FUNCTION_BLOCK AR_CALIBRATE_2P_REF (* Adapter-based 2-point calibration (Low/High, independently stored - no CO-before-CS style ordering dependency) - reference targets (Y_LOW/Y_HIGH) are live AR sockets, persisted via 2 additional AR2 plugs (LOW_REF/HIGH_REF), same live-echo pattern as AR_CALIBRATE_SQ_REF *)
  (* Standard: 61499-1 *)
  (* Version 1.3, 2026-09-21, Franz Höpfinger, Code-Review-Fund (PR #260): xClipping clippte bisher unconditional auf [LOW_REF,HIGH_REF], auch wenn nur EIN Punkt kalibriert war - der jeweils andere, noch unkalibrierte Referenzwert stand dann noch auf seinem INI_AR2-Default 0.0, wodurch der frisch eingefuehrte Partial-Kalibrierung-Fallback (Y.D1 := LOW_REF.DI1 bzw. HIGH_REF.DI1) sofort wieder auf 0.0 zurueckgeklemmt wurde - der Wert griff also weiterhin nicht sofort. Clipping jetzt zusaetzlich an xLowCal AND xHighCal gegated. *)
  (* Version 1.2, 2026-09-21, Franz Höpfinger, Genauso geaendert wie AR_CALIBRATE_3P_REF: INIT/QI/QO/INITO-Pattern (Enable/Disable) ergaenzt. Neuer Input xClipping (Default TRUE) - bisher clippte dieser Typ ueberhaupt nicht, jetzt optional auf LOW_REF..HIGH_REF klemmbar (FALSE = altes Verhalten, keine Klemmung). Neue interne Kalibriert-Flags xLowCal/xHighCal (latchen TRUE, sobald der jeweilige Rohwert vom INI_AR2-Default 0.0 abweicht): solange nur EIN Punkt kalibriert ist, wurde bisher trotzdem interpoliert - gegen einen Rohwert-Default von 0.0 fuer den jeweils anderen, noch unkalibrierten Punkt, was ein Garbage-Ergebnis lieferte. Jetzt liefert REQ in diesem Fall stattdessen direkt den REF-Wert des einen kalibrierten Punkts. *)
  (* Version 1.1, 2026-09-17, Franz Höpfinger, C_LOW/C_HIGH von AX-Sockets (mit [C_LOW.D1]/[C_HIGH.D1]-Flankenwaechter) auf reine EventInputs umgestellt - Franz: jeder echte Aufrufer (VT-Taste, OPC-UA-Methode, Remote-Toggle-Trigger nach Merge) liefert ohnehin ein atomares, einmaliges Event, der D1-Wert war bei jedem tatsaechlichen Caller immer hartcodiert TRUE (via AX_BOOL_TO_X) und der Guard filterte nie etwas - reine akademische Rechtfertigung ohne echten Nutzen. Aufrufer muessen jetzt direkt ein Event statt eines AX-Adapters anschliessen (AX_BOOL_TO_X-Umweg entfaellt). *)
  (* Version 1.0, 2026-09-11, Meisterschulen am Ostbahnhof, Ersatz fuer AR_CALIBRATE_SQ_REF: dieselbe Formel/dasselbe Ergebnis, aber ohne die CO-vor-CS-Abhaengigkeit - jeder Punkt speichert unabhaengig seinen Rohwert (wie AR_CALIBRATE_3P), die Interpolation passiert erst live bei X.E1, nicht mehr inkrementell beim Kalibrieren selbst. *)
  PACKAGE adapter::Engineering::measurements;
  (* Documentation:
  Formula
   Y = LOW_REF + (X - X_LOW) * (HIGH_REF - LOW_REF) / (X_HIGH - X_LOW), clipped to LOW_REF..HIGH_REF unless xClipping = FALSE Partial Calibration (before both points are set)
   Each point is tracked internally (xLowCal/xHighCal, latched TRUE once its raw value differs from the INI_AR2 default 0.0). Until both are calibrated, REQ falls back to the one already-known REF value instead of interpolating against the other point's still-0.0 default (which previously produced a garbage result as soon as only one side had been calibrated).
   Why this replaces AR_CALIBRATE_SQ_REF
   AR_CALIBRATE_SQ_REF computes OFFSET/SCALE incrementally (CO sets OFFSET from a live SCALE, CS then recomputes both from an internal X_LOW_INT/Y_LOW_INT captured by CO) - CS is only mathematically valid after CO has run at least once, which needed an ECC-enforced order to avoid a silent garbage-OFFSET calibration.
   This type stores X_LOW/X_HIGH completely independently (exactly like AR_CALIBRATE_3P/AR_CALIBRATE_3P_REF store X_MIN/X_MID/X_MAX) and only combines them into a line at read-time (REQ), which runs on every X.E1 regardless of calibration state. There is no data dependency between C_LOW and C_HIGH, so there is nothing an enforced order could protect against - both points can be (re-)calibrated in any order, independently, at any time.
   Calibration (Two-Point, Free Order)
    - Low (C_LOW): Apply low reference, set Y_LOW to desired output, trigger C_LOW → X_LOW := X
   - High (C_HIGH): Apply high reference, set Y_HIGH to desired output, trigger C_HIGH → X_HIGH := X
    Either point can be recalibrated on its own at any later time (e.g. re-trimming a drifted zero point) without repeating the other.
   Reference Targets (Y_LOW / Y_HIGH) are live AR Sockets
   Same live-echo mechanism as AR_CALIBRATE_SQ_REF: Y_LOW/Y_HIGH are bidirectional AR2 Sockets fed from an external VT/web reader, mirrored out through the AR2 Plugs LOW_REF/HIGH_REF for persistence (INI_AR2/NVS_AR2), and echoed back via LOW_REF.EI1/HIGH_REF.EI1 so a boot-restored value shows up on screen without the operator re-entering it.
  *)
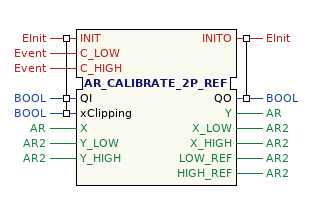
  EVENT_INPUT
    INIT : EInit WITH QI, xClipping; (* Initialization Request *)
    C_LOW; (* Calibrate Low Point - atomarer Trigger (VT-Taste/OPC-UA-Methode/Remote-Toggle nach Merge) *)
    C_HIGH; (* Calibrate High Point - atomarer Trigger (VT-Taste/OPC-UA-Methode/Remote-Toggle nach Merge) *)
  END_EVENT
  EVENT_OUTPUT
    INITO : EInit WITH QO; (* Initialization Confirm *)
  END_EVENT
  VAR_INPUT
    QI : BOOL; (* Input event qualifier *)
    xClipping : BOOL := TRUE; (* TRUE (Default) = Ausgang wird auf LOW_REF..HIGH_REF geklemmt; FALSE = kein Clipping, Extrapolation ueber die Kalibrierpunkte hinaus erlaubt (bisheriges Verhalten) *)
  END_VAR
  VAR_OUTPUT
    QO : BOOL; (* Output event qualifier *)
  END_VAR
  SOCKETS
    X : adapter::types::unidirectional::AR; (* Raw Input *)
    Y_LOW : adapter::types::bidirectional::AR2; (* Target output Y at the low calibration point - live edit in via EO1/DO1 (Socket-side swap), persisted/restored value echoed back out via EI1/DI1 for VT/web display *)
    Y_HIGH : adapter::types::bidirectional::AR2; (* Target output Y at the high calibration point - live edit in via EO1/DO1 (Socket-side swap), persisted/restored value echoed back out via EI1/DI1 for VT/web display *)
  END_SOCKETS
  PLUGS
    Y : adapter::types::unidirectional::AR; (* Calibrated Output *)
    X_LOW : adapter::types::bidirectional::AR2; (* Persisted raw input value at the low calibration point *)
    X_HIGH : adapter::types::bidirectional::AR2; (* Persisted raw input value at the high calibration point *)
    LOW_REF : adapter::types::bidirectional::AR2; (* Persisted low-point target reference (Y_LOW) *)
    HIGH_REF : adapter::types::bidirectional::AR2; (* Persisted high-point target reference (Y_HIGH) *)
  END_PLUGS
  VAR
    xLowCal : BOOL := FALSE; (* Latched TRUE sobald X_LOW.DI1 vom INI-Default 0.0 abweicht - LOW wurde mindestens einmal kalibriert (diese Session oder ueber Boot-Restore) *)
    xHighCal : BOOL := FALSE; (* Latched TRUE sobald X_HIGH.DI1 vom INI-Default 0.0 abweicht - HIGH wurde mindestens einmal kalibriert (diese Session oder ueber Boot-Restore) *)
  END_VAR
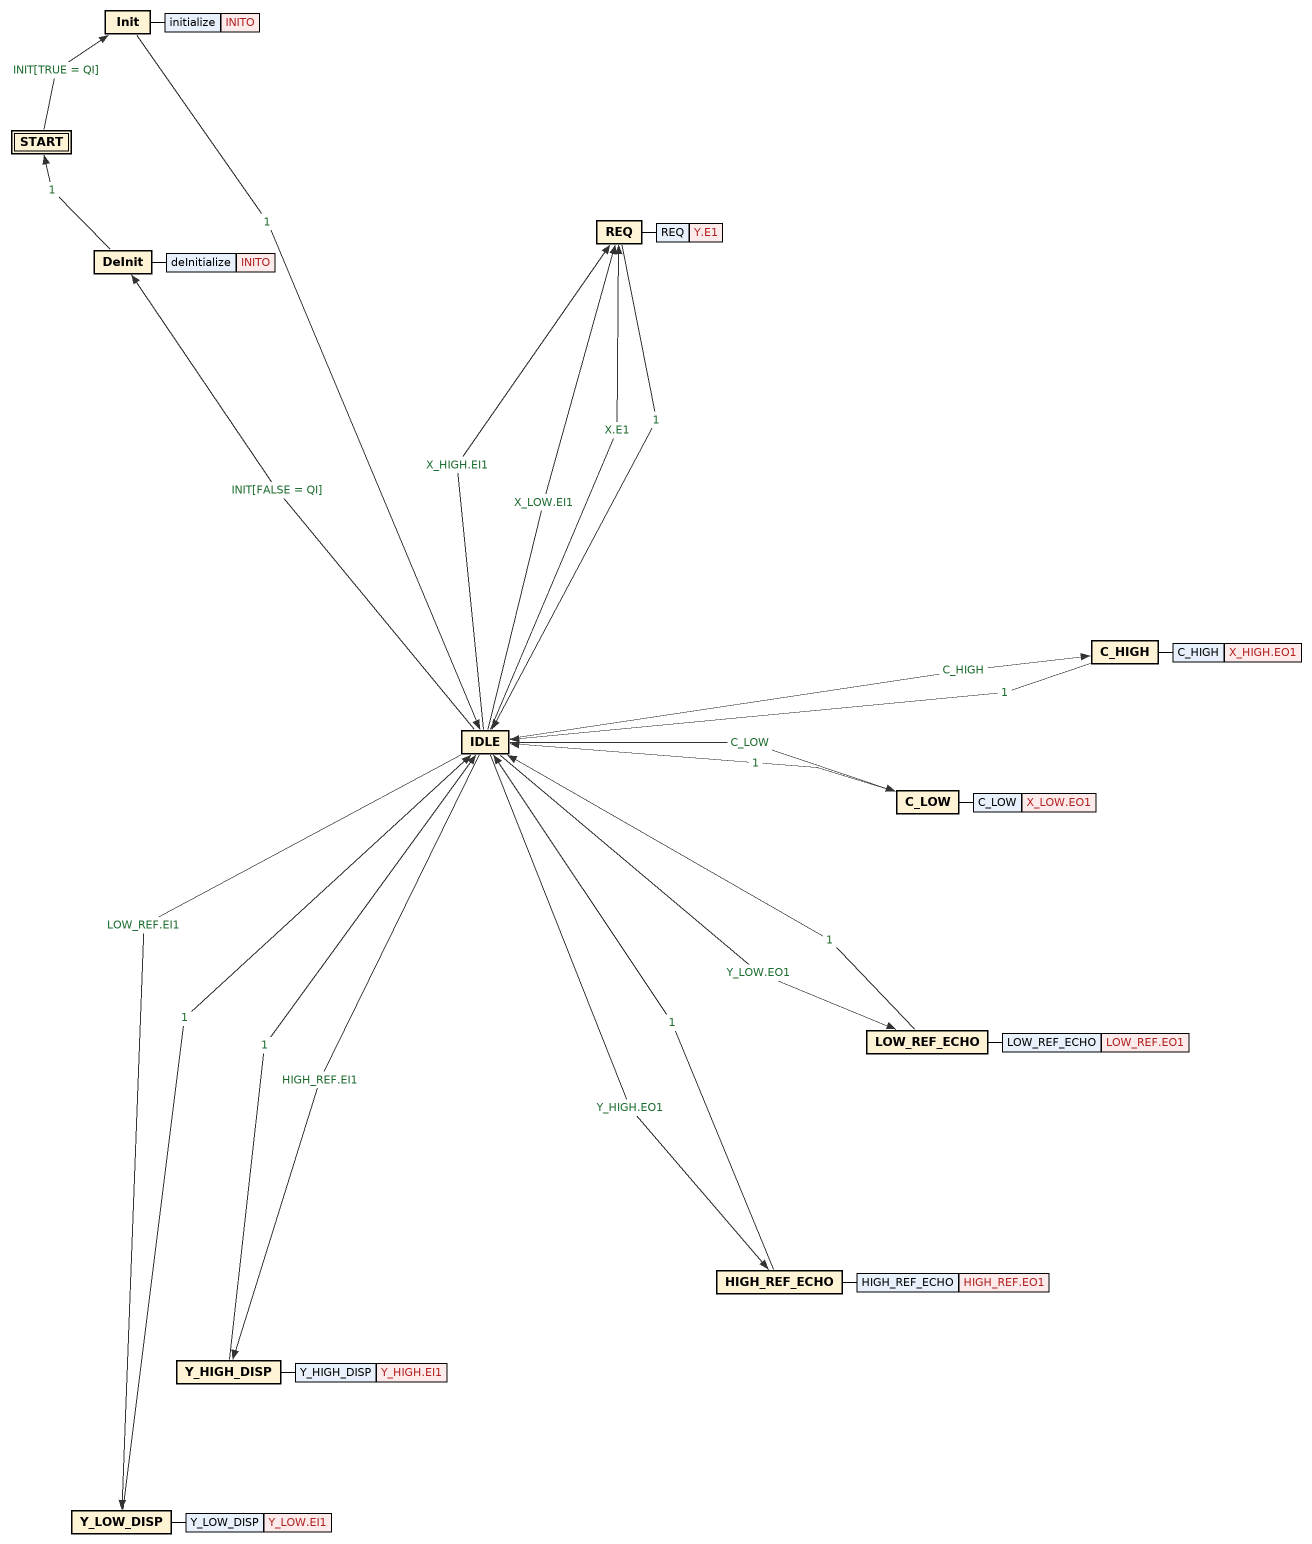
  EC_STATES
    START; (* Initial State *)
    Init : initialize -> INITO; (* Initialization *)
    DeInit : deInitialize -> INITO;
    IDLE;
    REQ : REQ -> Y.E1;
    C_LOW : C_LOW -> X_LOW.EO1;
    C_HIGH : C_HIGH -> X_HIGH.EO1;
    LOW_REF_ECHO : LOW_REF_ECHO -> LOW_REF.EO1;
    HIGH_REF_ECHO : HIGH_REF_ECHO -> HIGH_REF.EO1;
    Y_LOW_DISP : Y_LOW_DISP -> Y_LOW.EI1;
    Y_HIGH_DISP : Y_HIGH_DISP -> Y_HIGH.EI1;
  END_STATES
  EC_TRANSITIONS
    IDLE TO REQ := X.E1;
    REQ TO IDLE := 1;
    IDLE TO C_LOW := C_LOW;
    C_LOW TO IDLE := 1;
    IDLE TO C_HIGH := C_HIGH;
    C_HIGH TO IDLE := 1;
    IDLE TO REQ := X_LOW.EI1;
    IDLE TO REQ := X_HIGH.EI1;
    IDLE TO LOW_REF_ECHO := Y_LOW.EO1;
    LOW_REF_ECHO TO IDLE := 1;
    IDLE TO HIGH_REF_ECHO := Y_HIGH.EO1;
    HIGH_REF_ECHO TO IDLE := 1;
    IDLE TO Y_LOW_DISP := LOW_REF.EI1;
    Y_LOW_DISP TO IDLE := 1;
    IDLE TO Y_HIGH_DISP := HIGH_REF.EI1;
    Y_HIGH_DISP TO IDLE := 1;
    START TO Init := INIT[TRUE = QI];
    DeInit TO START := 1;
    Init TO IDLE := 1;
    IDLE TO DeInit := INIT[FALSE = QI];
  END_TRANSITIONS
  ALGORITHM initialize IN ST: (* Initialization algorithm *)
QO := QI;
  END_ALGORITHM
  ALGORITHM deInitialize IN ST: (* Normally executed algorithm *)
QO := FALSE;
  END_ALGORITHM
  ALGORITHM REQ IN ST: (* REQ *)
QO := QI;

IF TRUE = QI THEN
	(* latch "has been calibrated at least once" per point - a never-calibrated point stays
	 * exactly at the INI_AR2 DEFAULT_VALUE (0.0) forever, a real raw sensor value practically
	 * never is; a re-boot restores an already-calibrated point straight back to its non-0.0
	 * persisted value, so the latch stays correctly set across restarts *)
	IF X_LOW.DI1 <> 0.0 THEN xLowCal := TRUE; END_IF;
	IF X_HIGH.DI1 <> 0.0 THEN xHighCal := TRUE; END_IF;

	IF xLowCal AND xHighCal THEN
		(* both points calibrated - live linear interpolation, as before *)
		IF (X_HIGH.DI1 - X_LOW.DI1) <> 0.0 THEN
			Y.D1 := LOW_REF.DI1 + (X.D1 - X_LOW.DI1) * (HIGH_REF.DI1 - LOW_REF.DI1) / (X_HIGH.DI1 - X_LOW.DI1);
		ELSE
			Y.D1 := LOW_REF.DI1;
		END_IF;
	ELSIF xLowCal THEN
		(* only LOW calibrated so far - HIGH still at its 0.0 default, interpolating against it would
		 * give a garbage result, so fall back cleanly to the one REF value we actually have *)
		Y.D1 := LOW_REF.DI1;
	ELSIF xHighCal THEN
		Y.D1 := HIGH_REF.DI1;
	ELSE
		(* nothing calibrated yet *)
		Y.D1 := LOW_REF.DI1;
	END_IF;

	(* only clip once both bounding points are calibrated - otherwise the
	 * still-uncalibrated bound sits at its INI_AR2 default (0.0) and would
	 * clamp the partial-calibration fallback above right back to garbage *)
	IF xClipping AND xLowCal AND xHighCal THEN
		IF Y.D1 < LOW_REF.DI1 THEN
			Y.D1 := LOW_REF.DI1;
		ELSIF Y.D1 > HIGH_REF.DI1 THEN
			Y.D1 := HIGH_REF.DI1;
		END_IF;
	END_IF;
END_IF;
  END_ALGORITHM
  ALGORITHM C_LOW IN ST: (* Store current raw input as the low calibration point - independent of C_HIGH, repeatable any time *)
X_LOW.DO1 := X.D1;
  END_ALGORITHM
  ALGORITHM C_HIGH IN ST: (* Store current raw input as the high calibration point - independent of C_LOW, repeatable any time *)
X_HIGH.DO1 := X.D1;
  END_ALGORITHM
  ALGORITHM LOW_REF_ECHO IN ST: (* Persist live Y_LOW reference to INI *)
LOW_REF.DO1 := Y_LOW.DO1;
  END_ALGORITHM
  ALGORITHM HIGH_REF_ECHO IN ST: (* Persist live Y_HIGH reference to INI *)
HIGH_REF.DO1 := Y_HIGH.DO1;
  END_ALGORITHM
  ALGORITHM Y_LOW_DISP IN ST: (* Echo the persisted/restored LOW_REF value back out through Y_LOW for VT/web display (boot and after every change) *)
Y_LOW.DI1 := LOW_REF.DI1;
  END_ALGORITHM
  ALGORITHM Y_HIGH_DISP IN ST: (* Echo the persisted/restored HIGH_REF value back out through Y_HIGH for VT/web display (boot and after every change) *)
Y_HIGH.DI1 := HIGH_REF.DI1;
  END_ALGORITHM
END_FUNCTION_BLOCK
